// TIA Portal project "PID control" (V18)

(* hardware
DEVICE "S7-1200 station_1"  S7-1200 Station
   slot 0: "Rack_0"  S7-1200 Rack  Rack  V1.0
   slot 1: "PLC_1"  CPU 1217C DC/DC/DC  6ES7 217-1AG40-0XB0  V4.6
*)

// ===== PLC "PLC_1"  CPU 1217C DC/DC/DC =====

DATA_BLOCK "Batch_1"   // DB3
{ S7_Optimized_Access := 'TRUE' }
VERSION : 0.1
   VAR
      PID_MASTER_OUTPUT : Real;
      PID_MASTER_SETPOINT : Real;
      PID_MASTER_INPUT : Real;
      PID_SLAVE_INPUT : Real;
      PID_SLAVE_OUTHEAT : Real;
      PID_SLAVE_OUTCOOL : Real;
   END_VAR
BEGIN
END_DATA_BLOCK

DATA_BLOCK "LSim_I_DB"   // DB4
{ S7_Optimized_Access := 'TRUE' }
VERSION : 2.01
// stored: InstanceOfName LSim_I
"LSim_I"
BEGIN
END_DATA_BLOCK

DATA_BLOCK "LSim_IT1_DB"   // DB5
{ S7_Optimized_Access := 'TRUE' }
VERSION : 2.01
// stored: InstanceOfName LSim_IT1
"LSim_IT1"
BEGIN
END_DATA_BLOCK

DATA_BLOCK "LSim_PT3HeatCool_DB"   // DB6
{ S7_Optimized_Access := 'TRUE' }
VERSION : 2.01
// stored: InstanceOfName LSim_PT3HeatCool
"LSim_PT3HeatCool"
BEGIN
END_DATA_BLOCK

DATA_BLOCK "LSim_PT3_DB"   // DB7
{ S7_Optimized_Access := 'TRUE' }
VERSION : 2.01
// stored: InstanceOfName LSim_PT3
"LSim_PT3"
BEGIN
END_DATA_BLOCK

DATA_BLOCK "LSim_PT3HeatCool_DB_1"   // DB8
{ S7_Optimized_Access := 'TRUE' }
VERSION : 2.01
// stored: InstanceOfName LSim_PT3HeatCool
"LSim_PT3HeatCool"
BEGIN
END_DATA_BLOCK

FUNCTION_BLOCK "LSim_PT3"   // FB54, SCL
{ S7_Optimized_Access := 'TRUE' }
VERSION : 2.01
   VAR_INPUT
      input : Real;   // input variable
      tmLag1 : Real := 29.0;   // time lag 1 in s
      tmLag2 : Real := 17.5;   // time lag 2 in s
      tmLag3 : Real := 3.1;   // time lag 3 in s
      gain : Real := 1.0;   // proportional gain
      disturb : Real;   // disturbance variable (additional to "input")
      cycle : Real := 0.1;   // sample time [in sec]
      reset : Bool;   // complete restart (#output = #input)
   END_VAR
   VAR_OUTPUT
      error : Bool;   // error (#tmLag1 <= 0 or #tmLag2 <= 0 or #tmLag3 <= 0)
      status : Word;   // status (if #error = TRUE then status = 16#8001)
      output : Real;   // output signal (if #error = FALSE)
   END_VAR
   VAR
      statFback1 : Real;   // feedback path value 1
      statFback2 : Real;   // feedback path value 2
      statFback3 : Real;   // feedback path value 3
   END_VAR
   VAR_TEMP
      tempHvar : Real;   // help variable
      tempCycleR : Real;   // cycle to real
      tempTmLag1R : Real;   // time lag 1 to real
      tempTmLag2R : Real;   // time lag 2 to real
      tempTmLag3R : Real;   // time lag 3 to real
      tempOutvNew : Real;   // new output variable
   END_VAR
BEGIN
   //=============================================================================
   //SIEMENS AG
   //(c)Copyright 2017 All Rights Reserved
   //-----------------------------------------------------------------------------
   //Library:       Library for Controlled System Simulation
   //Tested with:   S7-1500 FW V2.0 / S7-1200 FW V4.2
   //Engineering:   STEP 7 V14 Upd2 (TIA Portal)
   //Restrictions:  Cyclic interrupt
   //Requirements:  memory card needed for S7-1500
   //Functionality: Simulation of an PT3-system
   //
   //                               gain
   //  F(p) = ------------------------------------------------------
   //         (tmLag1 * p + 1) * (tmLag2 * p + 1) * (tmLag3 * p + 1)
   //          
   //  Call the simulation in a cyclic interrupt with
   //  cyclic interrupt time at least = tmLag1/10!
   //-----------------------------------------------------------------------------
   //Change log table:
   //Version  Date       Expert in charge                Changes applied
   //02.00.00 03.02.2016 Siemens Industry Online Support Release (STEP 7 V13 SP1)
   //02.00.01 02.03.2017 Siemens Industry Online Support Release (STEP 7 V14)
   //=============================================================================
   // check parameter
   IF #tmLag1 <= 0 OR #tmLag2 <= 0 OR #tmLag3 <= 0 THEN
     #error := TRUE;
     #status := W#16#8001;     // Parameter Error
     #output := #input; //write output data
     #statFback1 := #input; //write static data
     #statFback2 := #input;
     #statFback3 := #input;
     RETURN;
   ELSE
     #error := FALSE;
     #status := W#16#0000;     // no error
   END_IF;

   IF #reset THEN //complete restart routine

     #output := #input;//write output data
     #statFback1 := #input;//write static data
     #statFback2 := #input;
     #statFback3 := #input;

   ELSE //cycle mode routine

     #tempCycleR  := #cycle*1000; //transform data type
     #tempTmLag1R := #tmLag1*1000;
     #tempTmLag2R := #tmLag2*1000;
     #tempTmLag3R := #tmLag3*1000;

     IF #tempCycleR * 0.5 > #tempTmLag1R THEN //limit TM_LAG1
       #tempTmLag1R := #tempCycleR * 0.5;
     END_IF;

     IF #tempCycleR * 0.5 > #tempTmLag2R THEN //limit TM_LAG2
       #tempTmLag2R := #tempCycleR * 0.5;
     END_IF;

     IF #tempCycleR * 0.5 > #tempTmLag3R THEN //limit TM_LAG2
       #tempTmLag3R := #tempCycleR * 0.5;
     END_IF;

     //1. first order lag algorithm
     #tempHvar     := #tempCycleR / (#tempTmLag1R * 2.0); 
     #tempHvar     := (#gain * (#input + #disturb) - #statFback1) * #tempHvar / (#tempHvar + 1.0);
     #tempOutvNew  := #tempHvar + #statFback1;
     #statFback1  := #tempHvar * 2.0 + #statFback1;

     //2. first order lag algorithm
     #tempHvar     := #tempCycleR / (#tempTmLag2R * 2.0); 
     #tempHvar     := ((#tempOutvNew - #statFback2) * #tempHvar) / (#tempHvar + 1.0);
     #tempOutvNew  := #tempHvar + #statFback2;
     #statFback2  := #tempHvar * 2.0 + #statFback2;

     //3. first order lag algorithm
     #tempHvar     := #tempCycleR / (#tempTmLag3R * 2.0); 
     #tempHvar     := ((#tempOutvNew - #statFback3) * #tempHvar) / (#tempHvar + 1.0);
     #tempOutvNew  := #tempHvar + #statFback3;
     #statFback3  := #tempHvar * 2.0 + #statFback3;

     #output := #tempOutvNew; //write output

   END_IF;
END_FUNCTION_BLOCK

FUNCTION_BLOCK "LSim_I"   // FB56, SCL
{ S7_Optimized_Access := 'TRUE' }
VERSION : 2.01
   VAR_INPUT
      calcParam : Bool;   // recalculate with new parameters
      input : Real;   // input signal
      tmLag1 : Real := 1.0;   // time constant T1 [sec]
      cycle : Real := 0.1;   // cyclic time [sec]
      maxOut : Real := 100.0;   // max. output limit
      minOut : Real;   // min. output limit
      reset : Bool;   // resets all relevant parameters to ‘0’ including the output
   END_VAR
   VAR_OUTPUT
      error : Bool;   // error (#tmLag1 <= 0)
      status : Word;   // status (if #tmLag1 <= 0 then status = 16#8001)
      maxReached : Bool;   // output has reached max. limit
      minReached : Bool;   // output has reached min. limit
      output : Real;   // output signal (if #error = FALSE)
   END_VAR
   VAR
      statRxn1 : Real;   // delayed input signal (n-1)
      statRyn1 : Real;   // delayed output signal (n-1)
      statRa1 : Real;
      statRb1 : Real;
      statOverfirst : Bool;
      statOutput : Real;   // output signal
   END_VAR
BEGIN
   //=============================================================================
   //SIEMENS AG
   //(c)Copyright 2017 All Rights Reserved
   //-----------------------------------------------------------------------------
   //Library:       Library for Controlled System Simulation
   //Tested with:   S7-1500 FW V2.0 / S7-1200 FW V4.2
   //Engineering:   STEP 7 V14 Upd2 (TIA Portal)
   //Restrictions:  Cyclic interrupt
   //Requirements:  memory card needed for S7-1500
   //Functionality: Simulation of a I-System
   //
   //             1
   //  F(p) = -----------
   //         (tmLag1*p)
   //          
   //  Call the simulation in a cyclic interrupt with
   //  cyclic interrupt time at least = tmLag1/10!
   //-----------------------------------------------------------------------------
   //Change log table:
   //Version  Date       Expert in charge                Changes applied
   //02.00.00 03.02.2016 Siemens Industry Online Support Release (STEP 7 V13 SP1)
   //02.00.01 02.03.2017 Siemens Industry Online Support Release (STEP 7 V14)
   //=============================================================================

   // check parameter
   IF #tmLag1 <= 0 THEN
     #error := True;
     #status := W#16#8001;     // Parameter Error
     #statRxn1 := 0.0;
     #statRyn1 := 0.0;
     #statOutput := 0;
     #output := 0;
     RETURN;
   ELSE
     #error := FALSE;
     #status := W#16#0000;     // no error
   END_IF;

   // calculates the z-parameter for the difference equatation
   IF #calcParam = True OR NOT #statOverfirst THEN
   #statOverfirst:=1;
     // Calculate z-parameters for IT1-System
   #statRb1 := #cycle/#tmLag1;
   #statRa1 := -1;

   END_IF;

   // reset Memory
   IF #reset = True THEN
     #statRxn1 := 0.0;
     #statRyn1 := 0.0;
     #statOutput:=0;
   END_IF;

   // save delayed output-signals
   #statRyn1:= #statOutput;

   // difference equatation for the I-system
   #statOutput := #statRxn1* #statRb1 - #statRyn1*#statRa1;

   // save delayed input-signals
   #statRxn1 := #input;

   // max limit of acutating variable
   IF #statOutput > #maxOut THEN
     #statOutput := #maxOut;
     #maxReached:= True;
   ELSE
     #maxReached := False;
   END_IF;

   // min limit of acutating variable
   IF #statOutput < #minOut THEN
     #statOutput := #minOut;
     #minReached := True;
   ELSE
     #minReached := False;
   END_IF;

   #output := #statOutput;
END_FUNCTION_BLOCK

FUNCTION_BLOCK "LSim_IT1"   // FB57, SCL
{ S7_Optimized_Access := 'TRUE' }
VERSION : 2.01
   VAR_INPUT
      calcParam : Bool;   // recalculate with new parameters
      input : Real;   // input signal
      tmLag1 : Real := 5.0;   // time constant T1 [sec]
      gain : Real := 1.0;   // gain factor
      cycle : Real := 0.1;   // cyclic time [sec]
      maxOut : Real := 100.0;   // max. output limit
      minOut : Real;   // min. output limit
      reset : Bool;   // resets all relevant parameters to ‘0’ including the output
   END_VAR
   VAR_OUTPUT
      error : Bool;   // error (#tmLag1 <= 0)
      status : Word;   // status (if #tmLag1 <= 0 then status = 16#8001)
      maxReached : Bool;   // output has reached max. limit
      minReached : Bool;   // output has reached min. limit
      output : Real;   // output signal (if #error = FALSE)
   END_VAR
   VAR
      statRxn2 : Real;   // delayed input signal (n-2)
      statRxn1 : Real;   // delayed input signal (n-1)
      statRyn2 : Real;   // delayed output signal (n-2)
      statRyn1 : Real;   // delayed output signal (n-1)
      statRf1 : Real;
      statRf2 : Real;
      statRe1 : Real;
      statRe2 : Real;
      statAlpha : Real;
      statOverfirst : Bool;
      statOutput : Real;   // output signal
   END_VAR
BEGIN
   //=============================================================================
   //SIEMENS AG
   //(c)Copyright 2017 All Rights Reserved
   //-----------------------------------------------------------------------------
   //Library:       Library for Controlled System Simulation
   //Tested with:   S7-1500 FW V2.0 / S7-1200 FW V4.2
   //Engineering:   STEP 7 V14 Upd2 (TIA Portal)
   //Restrictions:  Cyclic interrupt
   //Requirements:  memory card needed for S7-1500
   //Functionality: Simulation of a IT1-System
   //  
   //               gain
   //  F(p) = ------------------
   //         p * (tmLag1*p + 1)
   //         
   //  Call the simulation in a cyclic interrupt with
   //  cyclic interrupt time at least = tmLag1/10!
   //-----------------------------------------------------------------------------
   //Change log table:
   //Version  Date       Expert in charge                Changes applied
   //02.00.00 03.02.2016 Siemens Industry Online Support Release (STEP 7 V13 SP1)
   //02.00.01 02.03.2017 Siemens Industry Online Support Release (STEP 7 V14)
   //=============================================================================


   // check parameter
   IF #tmLag1 <= 0 THEN
     #error := True;
     #status := W#16#8001;     // Parameter Error
     #statRxn1 := 0.0;
     #statRyn1 := 0.0;
     #statRxn2 := 0.0;
     #statRyn2 := 0.0;
     #statOutput := 0;
     #output := 0;
     RETURN;
   ELSE
     #error := FALSE;
     #status := W#16#0000;     // no error
   END_IF;

   // calculates the z-parameter for the difference equatation
   IF #calcParam = True OR NOT #statOverfirst THEN
     #statOverfirst:=1;
   // calculates the z-parameter for the difference equatation of the IT1-System
   #statAlpha := EXP(-#cycle/#tmLag1);
   #statRe1 := -1 - #statAlpha;
   #statRe2 := #statAlpha;
   #statRf1 := #gain*(#cycle +(#statAlpha - 1)*#tmLag1);
   #statRf2 := #gain*(-#statAlpha*#cycle+(1-#statAlpha)*#tmLag1);
   END_IF;

   // reset Memory
   IF #reset = True THEN
     #statRxn1 := 0.0;
     #statRyn1 := 0.0;
     #statRxn2 := 0.0;
     #statRyn2 := 0.0;
     #statOutput:=0;
   END_IF;

   // save delayed output-signals
   #statRyn2:=#statRyn1;
   #statRyn1:= #statOutput;

   // difference equatation for IT1-System
   #statOutput := #statRxn1* #statRf1 + #statRxn2*#statRf2 - #statRyn1*#statRe1 - #statRyn2*#statRe2;

   // save delayed input-signals
   #statRxn2 := #statRxn1;
   #statRxn1 := #input;

   // max limit of acutating variable
   IF #statOutput > #maxOut THEN
   #statOutput := #maxOut;
   #maxReached := True;
   ELSE
     #maxReached := False;
   END_IF;

   // min limit of acutating variable
   IF #statOutput < #minOut THEN
     #statOutput := #minOut;
     #minReached := True;
   ELSE
     #minReached := False;
   END_IF;

   #output := #statOutput;
END_FUNCTION_BLOCK

FUNCTION_BLOCK "LSim_PT3HeatCool"   // FB64, SCL
{ S7_Optimized_Access := 'TRUE' }
VERSION : 2.01
   VAR_INPUT
      inputHeat : Real;   // input variable heating
      inputCool : Real;   // input variable cooling
      disturbHeat : Real;   // disturbance variable heating (additional to "inputHeat")
      disturbCool : Real;   // disturbance variable cooling (additional to "inputCool")
      ambTemp : Real := 20.0;   // ambient temperature
      gainHeat : Real := 1.5;   // proportional gain heating
      gainCool : Real := 3.0;   // proportional gain cooling
      tmLag1Heat : Real := 60.0;   // time lag 1 heating [s]
      tmLag2Heat : Real := 10.0;   // time lag 2 heating [s]
      tmLag3Heat : Real;   // time lag 3 heating [s]
      tmLag1Cool : Real := 60.0;   // time lag 1 cooling [s]
      tmLag2Cool : Real := 10.0;   // time lag 2 cooling [s]
      tmLag3Cool : Real;   // time lag 3 cooling [s]
      cycle : Real := 0.1;   // sample time [s]
   END_VAR
   VAR_OUTPUT
      output : Real;   // output variable
   END_VAR
   VAR_IN_OUT
      reset : Bool;   // complete restart
   END_VAR
   VAR
      statFback1 : Array[0..1] of Real;   // feedback value 1 heating/cooling
      statFback2 : Array[0..1] of Real;   // feedback value 2 heating/cooling
      statFback3 : Array[0..1] of Real;   // feedback value 3 heating/cooling
   END_VAR
   VAR_TEMP
      tempHvar : Real;   // helper
      tempCycleR : Real;   // sampling time
      tempTmLag1R : Real;   // delay time 1
      tempTmLag2R : Real;   // delay time 2
      tempTmLag3R : Real;   // delay time 3
      tempIndex : Int;   // control variable
      tempOutvNew : Array[0..1] of Real;   // new output value heating/cooling
   END_VAR
BEGIN
   //=============================================================================
   //SIEMENS AG
   //(c)Copyright 2017 All Rights Reserved
   //-----------------------------------------------------------------------------
   //Library:       Library for Controlled System Simulation
   //Tested with:   S7-1500 FW V2.0 / S7-1200 FW V4.2
   //Engineering:   STEP 7 V14 Upd2 (TIA Portal)
   //Restrictions:  Cyclic interrupt
   //Requirements:  memory card needed for S7-1500
   //Functionality: Simulation of an PT3-system with heating and cooling input
   //-----------------------------------------------------------------------------
   //Change log table:
   //Version  Date       Expert in charge                Changes applied
   //02.00.00 03.02.2016 Siemens Industry Online Support Release (STEP 7 V13 SP1)
   //02.00.01 02.03.2017 Siemens Industry Online Support Release (STEP 7 V14)
   //=============================================================================
   #tempOutvNew[0] := (#inputHeat + #disturbHeat) * #gainHeat;
   #tempOutvNew[1] := (#inputCool + #disturbCool) * #gainCool;

   IF #reset
   THEN
     //restart

     //write output parameters
     #output := #tempOutvNew[0] - #tempOutvNew[1] + #ambTemp;

     //write static local variables
     FOR #tempIndex := 0 TO 1 DO
       #statFback1[#tempIndex] := #tempOutvNew[#tempIndex];
       #statFback2[#tempIndex] := #statFback1[#tempIndex];
       #statFback3[#tempIndex] := #statFback2[#tempIndex];
     END_FOR;

     #reset := FALSE;
   ELSE
     //smoothing  
     #tempCycleR := #cycle;
     IF #tempCycleR < 0.001
     THEN
       //low limit sampling time
       #tempCycleR := 0.001;
     END_IF;

     FOR #tempIndex := 0 TO 1 DO

       IF #tempIndex = 0
       THEN
         #tempTmLag1R := #tmLag1Heat;
         #tempTmLag2R := #tmLag2Heat;
         #tempTmLag3R := #tmLag3Heat;
       ELSE
         #tempTmLag1R := #tmLag1Cool;
         #tempTmLag2R := #tmLag2Cool;
         #tempTmLag3R := #tmLag3Cool;
       END_IF;

       //1.delay
       IF #tempTmLag1R >= #tempCycleR * 0.5
       THEN
         #tempHvar := #tempCycleR / (2.0 * #tempTmLag1R + #tempCycleR);
         #tempHvar := (#tempOutvNew[#tempIndex] - #statFback1[#tempIndex]) * #tempHvar;
         //calculate new output value
         #tempOutvNew[#tempIndex] := #statFback1[#tempIndex] + #tempHvar;
         //calculate new feedback value
         #statFback1[#tempIndex] := #statFback1[#tempIndex] + 2.0 * #tempHvar;
       ELSE  //----------------------------------- implicit PT1
         #tempHvar := #tempCycleR / (#tempTmLag1R + #tempCycleR);
         //calculate new feedback value
         #statFback1[#tempIndex] := #statFback1[#tempIndex] + (#tempOutvNew[#tempIndex] - #statFback1[#tempIndex]) * #tempHvar;
         //calculate new output value
         #tempOutvNew[#tempIndex] := #statFback1[#tempIndex];
       END_IF;

       //2.delay heating
       IF #tempTmLag2R >= #tempCycleR * 0.5
       THEN
         #tempHvar := #tempCycleR / (2.0 * #tempTmLag2R + #tempCycleR);
         #tempHvar := (#tempOutvNew[#tempIndex] - #statFback2[#tempIndex]) * #tempHvar;
         //calculate new output value
         #tempOutvNew[#tempIndex] := #statFback2[#tempIndex] + #tempHvar;
         //calculate new feedback value
         #statFback2[#tempIndex] := #statFback2[#tempIndex] + 2.0 * #tempHvar;
       ELSE
         #statFback2[#tempIndex] := #tempOutvNew[#tempIndex];
       END_IF;

       //3.delay heating
       IF #tempTmLag3R >= #tempCycleR * 0.5
       THEN
         #tempHvar := #tempCycleR / (2.0 * #tempTmLag3R + #tempCycleR);
         #tempHvar := (#tempOutvNew[#tempIndex] - #statFback3[#tempIndex]) * #tempHvar;
         //calculate new output value
         #tempOutvNew[#tempIndex] := #statFback3[#tempIndex] + #tempHvar;
         //calculate new feedback value
         #statFback3[#tempIndex] := #statFback3[#tempIndex] + 2.0 * #tempHvar;
       ELSE
         #statFback3[#tempIndex] := #tempOutvNew[#tempIndex];
       END_IF;

     END_FOR;

     #output := #tempOutvNew[0] - #tempOutvNew[1] + #ambTemp;
   END_IF;
END_FUNCTION_BLOCK

ORGANIZATION_BLOCK "Main"   // OB1, LAD, ProgramCycle
TITLE = "Main Program Sweep (Cycle)"
{ S7_Optimized_Access := 'TRUE' }
VERSION : 0.1
   VAR_INPUT
      Initial_Call : Bool;   // Initial call of this OB
      Remanence : Bool;   // =True, if remanent data are available
   END_VAR
BEGIN

REGION Network 1
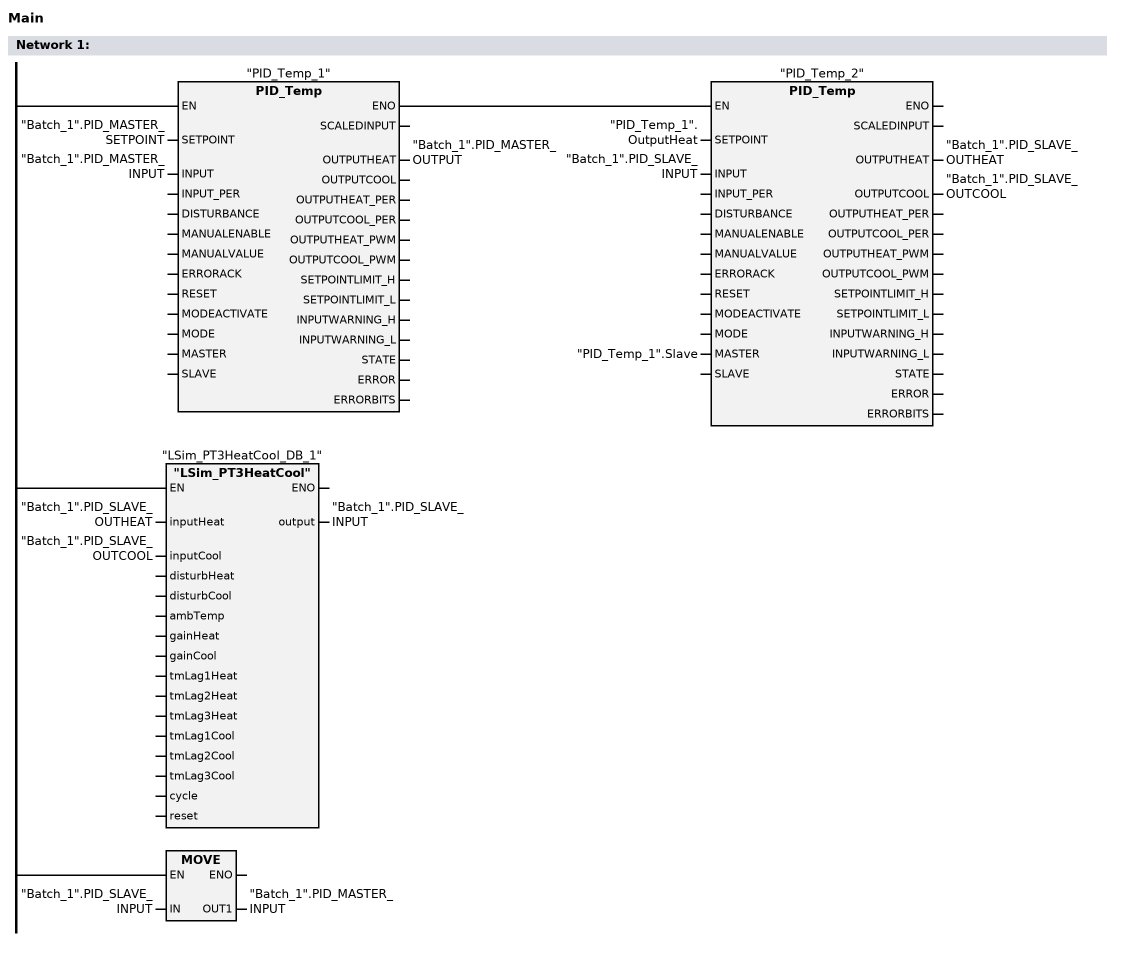
   // ENO of a box is taken as its EN; it also drops when the box reports an error
   "PID_Temp_1"(Setpoint := "Batch_1".PID_MASTER_SETPOINT,   // PID_Temp
                Input := "Batch_1".PID_MASTER_INPUT,
                OutputHeat => "Batch_1".PID_MASTER_OUTPUT);
   "PID_Temp_2"(Setpoint := "PID_Temp_1".OutputHeat,   // PID_Temp
                Input := "Batch_1".PID_SLAVE_INPUT,
                Master := "PID_Temp_1".Slave,
                OutputHeat => "Batch_1".PID_SLAVE_OUTHEAT,
                OutputCool => "Batch_1".PID_SLAVE_OUTCOOL);
   "LSim_PT3HeatCool_DB_1"(inputHeat := "Batch_1".PID_SLAVE_OUTHEAT,   // "LSim_PT3HeatCool"
                           inputCool := "Batch_1".PID_SLAVE_OUTCOOL,
                           output => "Batch_1".PID_SLAVE_INPUT);
   "Batch_1".PID_MASTER_INPUT := "Batch_1".PID_SLAVE_INPUT;
END_REGION
END_ORGANIZATION_BLOCK